TYPE T_JANSSEN_READING :
STRUCT
	Value:	LREAL;
END_STRUCT
END_TYPE

(* stored: Version 1.1.0.1, ProductVersion 3.1.4024.12
   DUT T_JANSSEN_READING: Id {d41027da-c930-4f58-8ff0-5fa8302d30f4} *)
